// TIA Portal V19 export
FUNCTION "DecoilersHU_CALL" : Void   // FC115, LAD
TITLE = DECOILERS HYDRAULIC UNIT CALL
// stored: SetENOAutomatically false
BEGIN

REGION Network 1: Data in
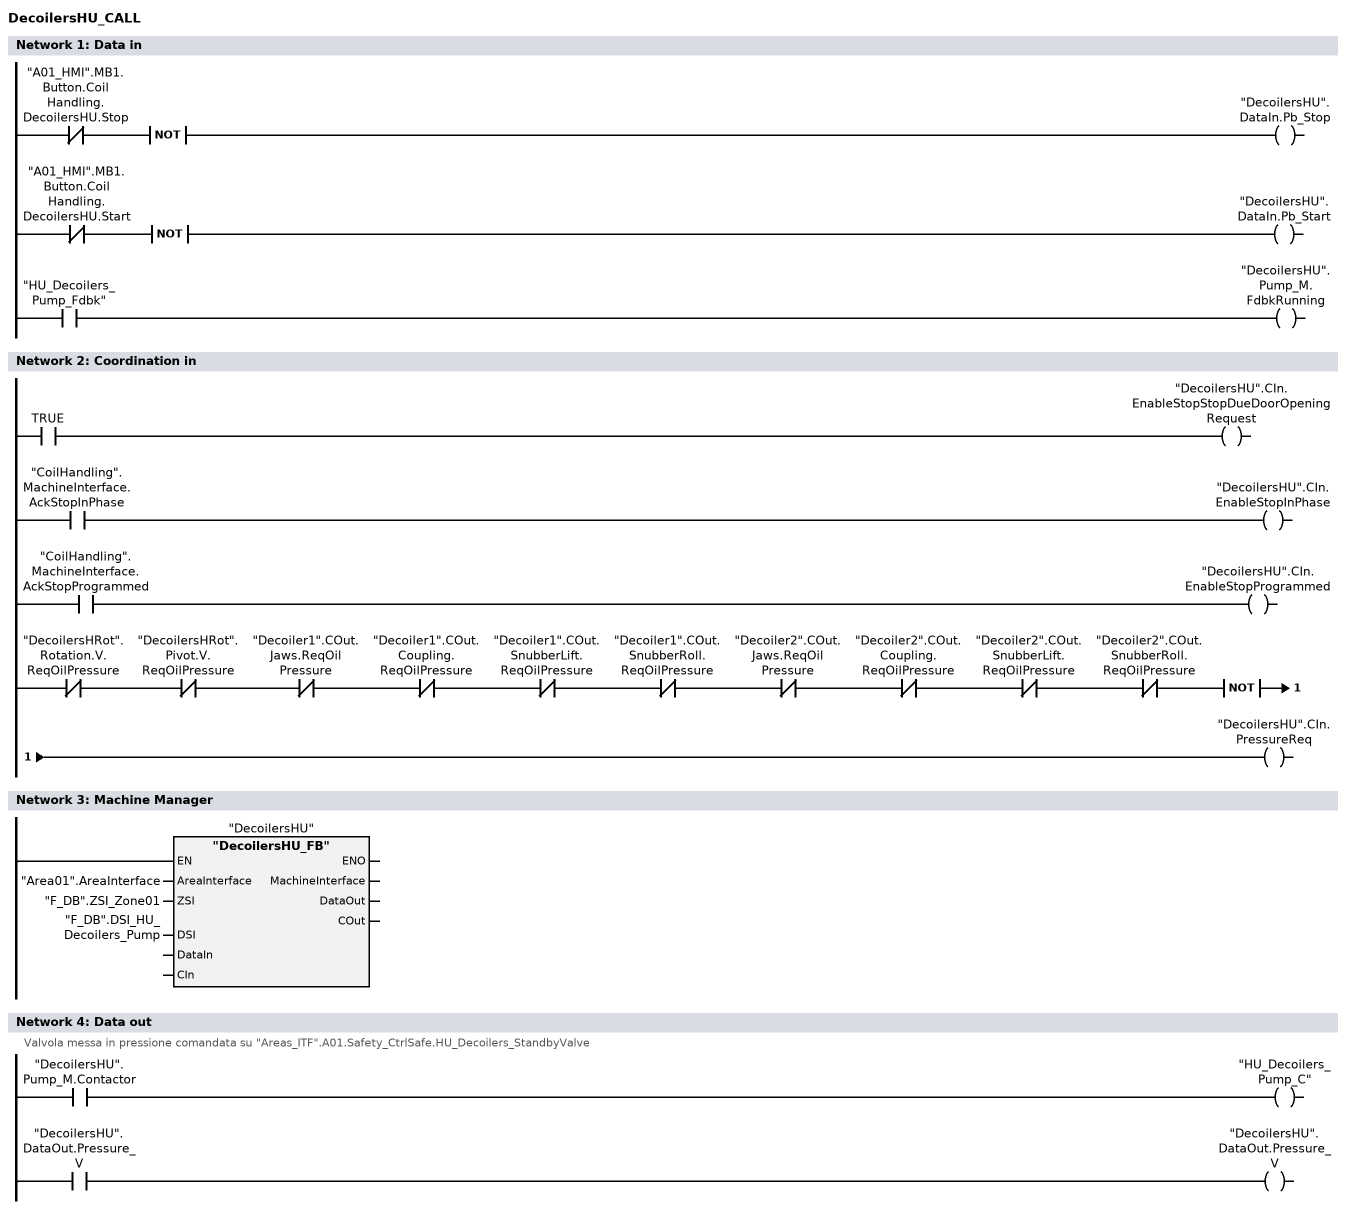
   RUNG wire#powerrail
      I_Contact( "A01_HMI".MB1.Button.CoilHandling.DecoilersHU.Stop )
      Not()
      Coil( "DecoilersHU".DataIn.Pb_Stop )
   END_RUNG
   RUNG wire#powerrail
      I_Contact( "A01_HMI".MB1.Button.CoilHandling.DecoilersHU.Start )
      Not()
      Coil( "DecoilersHU".DataIn.Pb_Start )
   END_RUNG
   RUNG wire#powerrail
      Contact( "HU_Decoilers_Pump_Fdbk" )
      Coil( "DecoilersHU".Pump_M.FdbkRunning )
   END_RUNG
   // the same network as SCL:
   "DecoilersHU".DataIn.Pb_Stop := NOT (NOT "A01_HMI".MB1.Button.CoilHandling.DecoilersHU.Stop);
   "DecoilersHU".DataIn.Pb_Start := NOT (NOT "A01_HMI".MB1.Button.CoilHandling.DecoilersHU.Start);
   "DecoilersHU".Pump_M.FdbkRunning := "HU_Decoilers_Pump_Fdbk";
END_REGION

REGION Network 2: Coordination in
   RUNG wire#powerrail
      Contact( TRUE )
      Coil( "DecoilersHU".CIn.EnableStopStopDueDoorOpeningRequest )
   END_RUNG
   RUNG wire#powerrail
      Contact( "CoilHandling".MachineInterface.AckStopInPhase )
      Coil( "DecoilersHU".CIn.EnableStopInPhase )
   END_RUNG
   RUNG wire#powerrail
      Contact( "CoilHandling".MachineInterface.AckStopProgrammed )
      Coil( "DecoilersHU".CIn.EnableStopProgrammed )
   END_RUNG
   RUNG wire#powerrail
      I_Contact( "DecoilersHRot".Rotation.V.ReqOilPressure )
      I_Contact( "DecoilersHRot".Pivot.V.ReqOilPressure )
      I_Contact( "Decoiler1".COut.Jaws.ReqOilPressure )
      I_Contact( "Decoiler1".COut.Coupling.ReqOilPressure )
      I_Contact( "Decoiler1".COut.SnubberLift.ReqOilPressure )
      I_Contact( "Decoiler1".COut.SnubberRoll.ReqOilPressure )
      I_Contact( "Decoiler2".COut.Jaws.ReqOilPressure )
      I_Contact( "Decoiler2".COut.Coupling.ReqOilPressure )
      I_Contact( "Decoiler2".COut.SnubberLift.ReqOilPressure )
      I_Contact( "Decoiler2".COut.SnubberRoll.ReqOilPressure )
      Not()
      Coil( "DecoilersHU".CIn.PressureReq )
   END_RUNG
   // the same network as SCL:
   "DecoilersHU".CIn.EnableStopStopDueDoorOpeningRequest := TRUE;
   "DecoilersHU".CIn.EnableStopInPhase := "CoilHandling".MachineInterface.AckStopInPhase;
   "DecoilersHU".CIn.EnableStopProgrammed := "CoilHandling".MachineInterface.AckStopProgrammed;
   "DecoilersHU".CIn.PressureReq := NOT (NOT "DecoilersHRot".Rotation.V.ReqOilPressure AND NOT "DecoilersHRot".Pivot.V.ReqOilPressure AND NOT "Decoiler1".COut.Jaws.ReqOilPressure AND NOT "Decoiler1".COut.Coupling.ReqOilPressure AND NOT "Decoiler1".COut.SnubberLift.ReqOilPressure AND NOT "Decoiler1".COut.SnubberRoll.ReqOilPressure AND NOT "Decoiler2".COut.Jaws.ReqOilPressure AND NOT "Decoiler2".COut.Coupling.ReqOilPressure AND NOT "Decoiler2".COut.SnubberLift.ReqOilPressure AND NOT "Decoiler2".COut.SnubberRoll.ReqOilPressure);
END_REGION

REGION Network 3: Machine Manager
   RUNG wire#powerrail
      "DecoilersHU"(AreaInterface := "Area01".AreaInterface, ZSI := "F_DB".ZSI_Zone01, DSI := "F_DB".DSI_HU_Decoilers_Pump, DataIn :=, CIn :=, MachineInterface =>, DataOut =>, COut =>)
   END_RUNG
   // the same network as SCL:
   "DecoilersHU"(AreaInterface := "Area01".AreaInterface,   // "DecoilersHU_FB"
                 ZSI := "F_DB".ZSI_Zone01,
                 DSI := "F_DB".DSI_HU_Decoilers_Pump);
END_REGION

REGION Network 4: Data out
   // Valvola messa in pressione comandata su "Areas_ITF".A01.Safety_CtrlSafe.HU_Decoilers_StandbyValve
   RUNG wire#powerrail
      Contact( "DecoilersHU".Pump_M.Contactor )
      Coil( "HU_Decoilers_Pump_C" )
   END_RUNG
   RUNG wire#powerrail
      Contact( "DecoilersHU".DataOut.Pressure_V )
      Coil( "DecoilersHU".DataOut.Pressure_V )
   END_RUNG
   // the same network as SCL:
   "HU_Decoilers_Pump_C" := "DecoilersHU".Pump_M.Contactor;
   "DecoilersHU".DataOut.Pressure_V := "DecoilersHU".DataOut.Pressure_V;
END_REGION
END_FUNCTION
